DATA_BLOCK "Itf"
{ S7_Optimized_Access := 'TRUE' }
VERSION : 0.1
NON_RETAIN
   VAR
      prendi : Bool;
      posa : Bool;
      accendiAsse : Bool;
      vaiAHomeAsse : Bool;
      pinzaAperta : Bool;
      pinzaChiusa : Bool;
      inPosAlta : Bool;
      inPosBassa : Bool;
      asseAcceso : Bool;
      asseReferenziato : Bool;
      errori : Bool;
      fineMissionePresa : Bool;
      fineMissionePosa : Bool;
      posizioneAttuale : Real;
   END_VAR


BEGIN

END_DATA_BLOCK

